{attribute 'GeneratedUsingTerminal: KL9900-0056'}
{attribute addProperty BoxType "KL9900-0056"}
{attribute addProperty Id "Channel_1AT %Q*Channel_2E0D480D0"}
{attribute addProperty CRC "104794512"}
{attribute addProperty Size "0"}
TYPE KL_063F0990 :
STRUCT
	{attribute addProperty Name "Channel_1"}
	Channel_1 : Channel_2E0D480D;
END_STRUCT
END_TYPE

(* stored: Version 1.2.0.0, ProductVersion 3.1.4024.9
   DUT KL_063F0990: Id {24b654b9-1e6d-4cd6-a74a-1445d53f0085} *)
